FUNCTION_BLOCK FB_CSL_MAIN
VAR_INPUT
	bEnable		:	BOOL;
END_VAR
VAR_IN_OUT
	stIn		:	ST_CSL_In;
	stParams	: 	ST_CSL_Params;
	stOut		:	ST_CSL_Out;
END_VAR
VAR_OUTPUT
	eStep	: E_Step;	//current step of the state machine
	eSubStep: E_Step;
	eErrStep : E_Step;  //step where an error was raised
	eErrSubStep: E_Step;
	nErrid	: DINT;		//error identification code
	nErrSubid	: DINT;
	
	bFbEnd	: BOOL;
END_VAR
VAR
	bInitialized	: BOOL;		//FB initialization
	eNewStep : E_Step;			//request for a new step
	bEntryact	: 	BOOL;		//step entry action performed
	
	fbSensor	: 	FB_MSF_Sensor;
	fbPiston	:	FB_MSF_Pistons;
	
	fbOscillator:	FB_Oscillator;
	
	bFbSensorEnd: BOOL;
	bFbPistonEnd: BOOL;
	
	
	
	nSlot : INT;
	
	bPause: BOOL	:= FALSE;
	
	bConveyorFree : BOOL;
END_VAR

(*Initialization of the FB_Sensor*)
IF NOT bInitialized THEN
	eNewStep := E_Step.NoStep;
	eStep := E_Step.MainStop;
	bEntryAct := FALSE;
	bFbEnd := FALSE;
	bInitialized := TRUE;
ELSE
	
	(*Preamble*)
	
	(*Forcing the Error State*)
	IF NOT bEnable THEN
		eNewStep := E_Step.NeOrError;
	END_IF	
	
	(*State change management*)
	IF eNewStep <> E_Step.NoStep THEN
		eStep := eNewStep;
		eNewStep := E_Step.NoStep;
		bEntryact := FALSE;
	END_IF
	
	IF stIn.bStop THEN
		bPause := TRUE;
	END_IF
	
	fbOscillator(enable := TRUE, t_high := T#500MS, t_low := T#500MS);

	(*Case*)
	CASE eStep OF
		
		(*MainStop Step - S0*)
		E_Step.MainStop :
			(*Body*)
			bPause := FALSE;
			
			stOut.bLStart	:= fbOscillator.q;
			stOut.bLStop := FALSE;
			stOut.bLAck := FALSE;
		
			(*Transition - to MainSensor*)
			IF stIn.bStart AND bEnable THEN
				eNewStep := E_Step.MainSensor;
			END_IF
			
			(*Exit Act*)
			IF eNewStep <> E_Step.NoStep THEN
				IF eNewStep = E_Step.NeOrError THEN
					eErrStep := eStep;
					//nErrId	:= 16#9999_9999;
				END_IF
			END_IF
			
		(*MainSensor Step - S1*)
		E_Step.MainSensor :
			(*Body*)
			stOut.bLStart	:= TRUE;
			IF bPause THEN
				stOut.bLStop := fbOscillator.q;
			ELSE
				stOut.bLStop := FALSE;
			END_IF
			stOut.bLAck := FALSE;
		
			fbSensor(
				stIn:= stIn, 
				bEnable:= bEnable, 
				eStep=> eSubStep, 
				eErrStep=> eErrSubStep, 
				nErrId=> nErrSubId,
				bFbEnd=> bFbSensorEnd, 
				stOut:= stOut, 
				nSlot=> nSlot, 
				stParams:= stParams
			);
			
			(*Transition - to Processing*)
			IF bFbSensorEnd AND bEnable THEN
				eNewStep := E_Step.MainPiston;
			END_IF
			
			(*Exit Act*)
			IF eNewStep <> E_Step.NoStep THEN
				IF eNewStep = E_Step.NeOrError THEN
					eErrStep := eStep;
					//nErrId	:= 16#9999_9999;
				END_IF
			END_IF
		
		(*MainPiston Step - S2*)
		E_Step.MainPiston :
			(*Body*)
			stOut.bLStart	:= TRUE;
			IF bPause THEN
				stOut.bLStop := fbOscillator.q;
			ELSE
				stOut.bLStop := FALSE;
			END_IF
			stOut.bLAck := FALSE;
		
			fbPiston(
				bEnable:= bEnable, 
				slot:= nSlot, 
				stIn:= stIn, 
				stParams:= stParams, 
				stOut:= stOut, 
				eStep=> eSubStep, 
				eErrStep=> eErrSubStep, 
				nErrid=> nErrSubId, 
				bFbEnd=> bFbPistonEnd
			);
			
			(*Transition - to MainSensor*)
			IF bFbPistonEnd AND bEnable THEN
				eNewStep := E_Step.MainSensor;
			END_IF
			
			(*Transition - to MainPause*)
			IF bPause AND bEnable THEN
				eNewStep := E_Step.MainPause;
			END_IF
			
			(*Exit Act*)
			IF eNewStep <> E_Step.NoStep THEN
				IF eNewStep = E_Step.NeOrError THEN
					eErrStep := eStep;
					//nErrId	:= 16#9999_9999;
				END_IF
			END_IF	
			
		(*MainPause Step - S3*)
		E_Step.MainPause :
			(*Body*)
			stOut.bLStart	:= FALSE;
			stOut.bLStop := TRUE;
			stOut.bLAck := FALSE;
			
			(*Transition - to MainSensor*)
			IF stIn.bStart AND bEnable THEN
				eNewStep := E_Step.MainSensor;
				bPause := FALSE;
			END_IF
			
			(*Exit Act*)
			IF eNewStep <> E_Step.NoStep THEN
				IF eNewStep = E_Step.NeOrError THEN
					eErrStep := eStep;
					//nErrId	:= 16#9999_9999;
				END_IF
			END_IF	
		
		(*MainEmergency Step - S4*)
		E_Step.MainEmergency :	
			(*Body*)
			stOut.bLStart	:= FALSE;
			stOut.bLStop := FALSE;
			stOut.bLAck := fbOscillator.q;
			
			
			//da vedere il pilotaggio delle uscite: motore, compressore e valvole
			stOut.bMotor := FALSE;
		
			(*Transition - to Measuring*)
			IF stIn.bAck AND bEnable THEN
				eNewStep := E_Step.MainAcknowledge;
			END_IF
			
			(*Exit Act*)
			IF eNewStep <> E_Step.NoStep THEN
				IF eNewStep = E_Step.NeOrError THEN
					eErrStep := eStep;
					//nErrId	:= 16#9999_9999;
				END_IF
			END_IF
			
		(*MainAcknowledge Step - S5*)	
		E_Step.MainAcknowledge :		
			(*Body*)
			stOut.bLStart	:= FALSE;
			stOut.bLStop := FALSE;
			stOut.bLAck := TRUE;
			
			//fb per liberare il nastro
				
		
			(*Transition - to Measuring*)
			IF bConveyorFree AND bEnable THEN
				eNewStep := E_Step.MainStop;
			END_IF
			
			(*Exit Act*)
			IF eNewStep <> E_Step.NoStep THEN
				IF eNewStep = E_Step.NeOrError THEN
					eErrStep := eStep;
					//nErrId	:= 16#9999_9999;
				END_IF
			END_IF
		
		(*NeOrError step*)	
		E_Step.NeOrError :
			(*Body*)
			stOut.bLStart	:= fbOscillator.q;
			stOut.bLStop := fbOscillator.q;
			stOut.bLAck := fbOscillator.q;
			
			stOut.bMotor := FALSE;
		
			(*Transition - to Measuring*)
			
			
			(*Exit Act*)
			IF eNewStep <> E_Step.NoStep THEN
				IF eNewStep = E_Step.NeOrError THEN
					eErrStep := eStep;
					//nErrId	:= 16#9999_9999;
				END_IF
			END_IF
			
	END_CASE
END_IF

END_FUNCTION_BLOCK

(* stored: Version 1.1.0.1, ProductVersion 3.1.4024.12
   POU FB_CSL_MAIN: Id {f7c0fb49-0a9a-4d93-8227-9668f0bcf9c2}, SpecialFunc None *)
